// TIA Portal V18 export
DATA_BLOCK "SIM_VALVE"   // DB29
{ S7_Optimized_Access := 'FALSE' }
VERSION : 0.1
// stored: AutoNumber true, DBAccessibleFromOPCUA true, DBAccessibleFromWebserver true, IsOnlyStoredInLoadMemory false, IsWriteProtectedInAS false
   VAR
      "H/SSR_019_XV01_CLOSEFB" : Bool;
      "H/SSR_019_XV02_OPENFB" : Bool;
      "H/SSR_019_XV02_CLOSEFB" : Bool;
      "H/SSR_019_XV03_OPENFB" : Bool;
      "H/SSR_019_XV03_CLOSEFB" : Bool;
      "H/SSR_019_XV04_CLOSEFB" : Bool;
      "H/SSR_019_XV04_OPENFB" : Bool;
      "H/SSR_019_XV05_OPENFB" : Bool;
      "H/SSR_019_XV05_CLOSEFB" : Bool;
      "H/SSR_019_XV06_OPENFB" : Bool;
      "H/SSR_019_XV06_CLOSEFB" : Bool;
      "H/SSR_019_XV07_OPENFB" : Bool;
      "H/SSR_019_XV07_CLOSEFB" : Bool;
      "H/SSR_019_XV08_OPENFB" : Bool;
      "H/SSR_019_XV08_CLOSEFB" : Bool;
      "H/SSR_019_XV09_OPENFB" : Bool;
      "H/SSR_019_XV09_CLOSEFB" : Bool;
      "H/SSR_019_XV10_OPENFB" : Bool;
      "H/SSR_019_XV10_CLOSEFB" : Bool;
      "H/SSR_019_XV11_OPENFB" : Bool;
      "H/SSR_019_XV11_CLOSEFB" : Bool;
      "H/SSR_019_XV12_OPENFB" : Bool;
      "H/SSR_019_XV12_CLOSEFB" : Bool;
      "H/SSR_019_XV13_OPENFB" : Bool;
      "H/SSR_019_XV13_CLOSEFB" : Bool;
      "H/SSR_019_TT01_IN" : Int;
      "H/SSR_019_TT02_IN" : Int;
      "H/SSR_019_APT01_IN" : Int;
      "H/SSR_019_GPT101_IN" : Int;
      "H/SSR_019_GPT201_IN" : Int;
      "H/SSR_019_GPT301_IN" : Int;
      "H/SSR_019_GPT401_IN" : Int;
      "H/SSR_019_GPT501_IN" : Int;
      "H/SSR_019_GPT601_IN" : Int;
      "H/SSR_019_TT03_IN" : Int;
      "H/SSR_019_TT01_PV" : Int;
      "H/SSR_019_XV01_OPENFB" : Bool;
      "H/SSR_019_TT02_INpv" : Bool;
      "H/SSR_019_APT01_PV" : Bool;
      "H/SSR_019_GPT101_PV" : Bool;
      "H/SSR_019_GPT201_PV" : Bool;
      "H/SSR_019_GPT301_PV" : Bool;
      "H/SSR_019_GPT401_PV" : Bool;
      "H/SSR_019_GPT501_PV" : Bool;
      "H/SSR_019_GPT601_PV" : Bool;
      "H/SSR_019_TT03_PV" : Bool;
      "H/SSR_019_TT01_PV_1" : Bool;
   END_VAR
BEGIN
END_DATA_BLOCK
